(* CODESYS project FB_TESTING.xml

Project tree, tasks and I/O mapping:
  program FB_TESTING [FBD]
*)

// FB_TESTING
PROGRAM FB_TESTING
(***********************************************************************************************
Object Name	: PLC_SUPPLY
Descrition	: Program to control the System Supply Switch to ensure the PLC turns OFF when the ignition turns OFF.
Author		: KP
Date		: 17/06/25
Rev			: P1
***********************************************************************************************)
VAR CONSTANT
	uiMinVoltage 		: UINT := 5000;    // Minimum Voltage in mV
END_VAR
VAR
	fbSystemSupply 	: ifmIOcommon.SystemSupply; // Function Block to monitor supply voltage on VBB15 (from ignition)
	fbSupplySwitch 	: ifmIOcommon.SupplySwitch; // Function Block to turn ON/OFF latching switch on VBB15 supply (from ignition)
	uiCurrSupplyVolt	: UINT ;    // Operating Voltage in mV
	TOF_0: TOF;
	Test: BOOL;
	dude: BOOL;
	fbenable: TON;
	xResult : BOOL;
	xTimerDone : BOOL;
END_VAR
VAR // added by the converter: edge detectors and wires of the graphical bodies
    _w1 : BOOL;
END_VAR

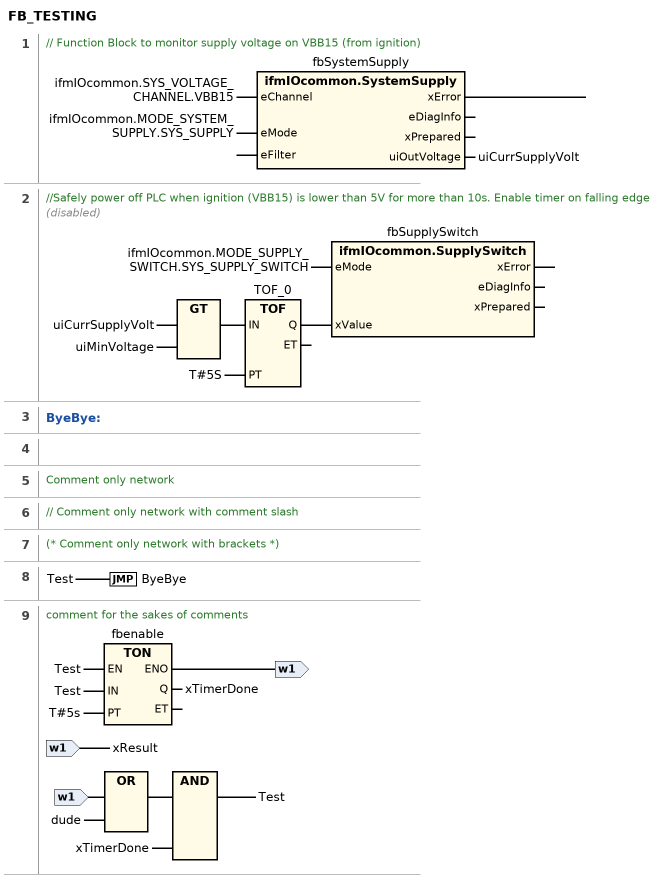
// NETWORK 1
// // Function Block to monitor supply voltage on VBB15 (from ignition)
fbSystemSupply(
    eChannel := ifmIOcommon.SYS_VOLTAGE_CHANNEL.VBB15,
    eMode := ifmIOcommon.MODE_SYSTEM_SUPPLY.SYS_SUPPLY,
    uiOutVoltage => uiCurrSupplyVolt); // ifmIOcommon.SystemSupply

// NETWORK 2 (disabled)
// //Safely power off PLC when ignition (VBB15) is lower than 5V for more than 10s. Enable timer on falling edge
// TOF_0(IN := uiCurrSupplyVolt > uiMinVoltage, PT := T#5S); // TOF
// fbSupplySwitch(eMode := ifmIOcommon.MODE_SUPPLY_SWITCH.SYS_SUPPLY_SWITCH, xValue := TOF_0.Q); // ifmIOcommon.SupplySwitch

// NETWORK 3
ByeBye: ;

// NETWORK 4

// NETWORK 5
// Comment only network

// NETWORK 6
// // Comment only network with comment slash

// NETWORK 7
// (* Comment only network with brackets *)

// NETWORK 8
IF Test THEN JMP ByeBye; END_IF

// NETWORK 9
// comment for the sakes of comments
_w1 := Test;
IF _w1 THEN
    fbenable(IN := Test, PT := T#5s, Q => xTimerDone); // TON
END_IF
xResult := _w1;
Test := (_w1 OR dude) AND xTimerDone;

END_PROGRAM
